TYPE EncoderTypeClass :
(
    NoEncoder          := 0,
    IncrementalEncoder := 1,
    AbsoluteEncoder    := 2
):= NoEncoder;
END_TYPE

(* stored: Version 1.1.0.1, ProductVersion 3.1.4024.0
   DUT EncoderTypeClass: Id {66179a35-7b0c-4440-b8bf-378ba0f6862b} *)
